Fanuc KAREL source: kt00161.KL

-- PROVISIONAL review KL for V1013-1; original PC SHA256 36df9140e1ac2d9f1c10a9cbb14354f69cc82e9566d54e5ff34b82de418ee9fc
-- Incomplete behavior may be omitted. Consult companion uncertainty JSON. Do not deploy.
PROGRAM KT00161
%NOLOCKGROUP
VAR
  I1 : INTEGER
  I2 : INTEGER
  OUT : INTEGER
BEGIN
  -- UNRESOLVED_PC offsets 5-16; opcodes 2E,23
  -- UNRESOLVED_PC offsets 21-32; opcodes 2E,23
  -- UNRESOLVED_PC offsets 37-48; opcodes 2E,23
  -- UNRESOLVED_PC offsets 53-64; opcodes 2E,23
  -- UNRESOLVED_PC offsets 69-88; opcodes 21,21,56,23
  -- UNRESOLVED_PC offsets 93-97; opcodes 7F
END KT00161
